FUNCTION_BLOCK ConveyorManualIProv (* Conveyor Manual Interface Provider *)
  (* Standard: 61499-2 *)
  (* Version 0.2, 2003-12-05, JHC, Rockwell Automation, Renamed from NEWCOMPFB. *)
  (* Version 0.1, 2002-01-08, JHC, Rockwell Automation, Added DLY FB as example. *)
  (* Version 0.0, 2000-05-27, JHC, Rockwell Automation *)
  (* Compiler header: package fb.rt.dasdA1.A2.Conveyor; *)
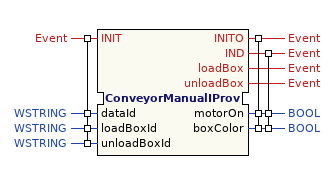
  EVENT_INPUT
    INIT WITH dataId, loadBoxId, unloadBoxId; (* Initialization Request *)
  END_EVENT
  EVENT_OUTPUT
    INITO WITH motorOn, boxColor; (* Initialization Confirm *)
    IND WITH motorOn, boxColor;
    loadBox;
    unloadBox;
  END_EVENT
  VAR_INPUT
    dataId : WSTRING;
    loadBoxId : WSTRING;
    unloadBoxId : WSTRING;
  END_VAR
  VAR_OUTPUT
    motorOn : BOOL;
    boxColor : BOOL;
  END_VAR
  FBS
    unloadBoxSub : SUBL_0;
    loadBoxSub : SUBL_0;
    data : SUBL_2;
  END_FBS
  EVENT_CONNECTIONS
    INIT TO data.INIT;
    loadBoxSub.IND TO loadBox;
    unloadBoxSub.IND TO unloadBox;
    loadBoxSub.INITO TO unloadBoxSub.INIT;
    data.INITO TO loadBoxSub.INIT;
    data.IND TO IND;
    unloadBoxSub.INITO TO INITO;
  END_CONNECTIONS
  DATA_CONNECTIONS
    loadBoxId TO loadBoxSub.ID;
    unloadBoxId TO unloadBoxSub.ID;
    dataId TO data.ID;
    data.RD_1 TO motorOn;
    data.RD_2 TO boxColor;
  END_CONNECTIONS
END_FUNCTION_BLOCK
